// Mitsubishi GX Works2 project: LRI   PLC: Q03UDV
// HelloWorld

PROGRAM MAIN
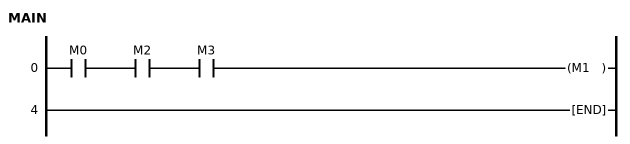
0     LD      M0
      AND     M2
      AND     M3
      OUT     M1
4     END
END_PROGRAM
